// TIA Portal V20 export
// export: Created 2025-12-01T14:57:06.1512195Z, ExportSetting None, DisplayName Totally Integrated Automation Portal, DisplayVersion V20 Update 3, DisplayName TIA Portal Openness, DisplayVersion V20 Update 3, DisplayName TIA Portal Version Control Interface, DisplayVersion V20 Update 3, DisplayName STEP 7 Professional, DisplayVersion V20 Update 3, DisplayName STEP 7 Safety, DisplayVersion V20 Update 2, DisplayName WinCC Basic/Comfort/Advanced, DisplayVersion V20 Update 3, DisplayName WinCC Professional, DisplayVersion V20 Update 3, DisplayName WinCC Unified, DisplayVersion V20 Update 3
FUNCTION "FC903_Tratamiento_MesasDeZona" : Void   // FC903, STL
{ S7_Optimized_Access := 'FALSE' }
// stored: AutoNumber false
   VAR_INPUT
      NumZona : UInt;
   END_VAR
   VAR_IN_OUT
      MesasDeZona : "InternasDeLaZona";
   END_VAR
   VAR_TEMP
      Zona : UInt;
      Mesa : UInt;
      MaxMesas : UInt;
      MesasParo : Bool;
      MesasBlando : Bool;
      MesasManual : Bool;
      MesasError : Bool;
      MesasTodasParo : Bool;
      MesasTodasManual : Bool;
   END_VAR
BEGIN

NETWORK
TITLE = Inicializacion
/////////////////////////////////////////////////////////////////////////////
/////////////////////////////////////////////////////////////////////////////
// --- Tareas Iniciales

      L     #NumZona;  // - Numero de Zana
      T     #Zona;

      L     #Zona;  // Es el CCPIF ?
      L     0;
      <>I;
      JC    CBOX;
      JU    CBOX;  // Para Tramiento el CBOX y CCPIF el mismo

/////////////////////////////////////////////////////////////////////////////
/////////////////////////////////////////////////////////////////////////////
// Es de Tipo CCPIF
CCPIF:NOP   0;
      SET;  // - Inicializar Variables Internas
      R     #MesasParo;  //   Para el CCPIF
      R     #MesasBlando;
      R     #MesasManual;
      R     #MesasError;
      R     #MesasTodasParo;
      R     #MesasTodasManual;
      JU    Final;  //   Finaliza para CCPIF


/////////////////////////////////////////////////////////////////////////////
/////////////////////////////////////////////////////////////////////////////
// Es de tipo CBOX
CBOX: NOP   0;

      SET;  // - Inicializar Variables Internas
      R     #MesasParo;  //   Para un CBOX
      R     #MesasBlando;
      R     #MesasManual;
      R     #MesasError;
      S     #MesasTodasParo;
      S     #MesasTodasManual;


/////////////////////////////////////////////////////////////////////////////
/////////////////////////////////////////////////////////////////////////////
// --- Datos iniciales de Trabajo

      L     "CTE_MaxMesas";  // - Numero Max. de Mesas en el PLC
      T     #MaxMesas;



NETWORK
TITLE = Tratamiento
/////////////////////////////////////////////////////////////////////////////
/////////////////////////////////////////////////////////////////////////////
// ---  Tratamiento del Estado de las Mesas que pertenecn a la Mesa

      L     1;  // Inicializar
      T     #Mesa;
InicioBucle:NOP   0;

      SET;  //    Zona 0
      L     "DB914_Conf_Mesas_DeZona".MesasDeZona[#Mesa, 0].ZonaPerteneceMesa;
      L     #Zona;
      ==I;
      JC    MesaEncontrada;

      SET;  //    Zona 1
      L     "DB914_Conf_Mesas_DeZona".MesasDeZona[#Mesa, 1].ZonaPerteneceMesa;
      L     #Zona;
      ==I;
      JC    MesaEncontrada;

      SET;  //    Zona 2
      L     "DB914_Conf_Mesas_DeZona".MesasDeZona[#Mesa, 2].ZonaPerteneceMesa;
      L     #Zona;
      ==I;
      JC    MesaEncontrada;

      SET;  //    Zona 3
      L     "DB914_Conf_Mesas_DeZona".MesasDeZona[#Mesa, 3].ZonaPerteneceMesa;
      L     #Zona;
      ==I;
      JC    MesaEncontrada;

      SET;  //    Zona 4
      L     "DB914_Conf_Mesas_DeZona".MesasDeZona[#Mesa, 4].ZonaPerteneceMesa;
      L     #Zona;
      ==I;
      JC    MesaEncontrada;

      JU    ContinuarBucle;


/////////////////////////////////////////////////////////////////////////////
/////////////////////////////////////////////////////////////////////////////
// --- Comprobacion del Estado Zona de la Mesa
MesaEncontrada:NOP   0;

      SET;  // - Alguna mesa en Error
      A     "DB902_Estado_ZonaMesa".EstadoMesas[#Mesa].Error_CBx;
      S     #MesasError;

      SET;  // - Alguna mesa en Paro
      AN    "DB902_Estado_ZonaMesa".EstadoMesas[#Mesa].Marcha_CBx;
      S     #MesasParo;

      SET;  // - Alguna mesa en ParoBlando
      A     "DB902_Estado_ZonaMesa".EstadoMesas[#Mesa].ParoBlando_CBx;
      S     #MesasBlando;

      SET;  // - Alguna mesa en Manual
      AN    "DB902_Estado_ZonaMesa".EstadoMesas[#Mesa].Automatico_CBx;
      S     #MesasManual;

      SET;  // - Todas las mesas en Paro
      A     "DB902_Estado_ZonaMesa".EstadoMesas[#Mesa].Marcha_CBx;
      R     #MesasTodasParo;

      SET;  // - Todas las mesas en Manual
      A     "DB902_Estado_ZonaMesa".EstadoMesas[#Mesa].Automatico_CBx;
      R     #MesasTodasManual;


/////////////////////////////////////////////////////////////////////////////
/////////////////////////////////////////////////////////////////////////////
// --- Comprobacion del Estado Zona de la Maquina

      SET;  // - Alguna Maquina en Error
      A     "DB903_Estado_ZonaMaquina".EstadoMaquina[#Mesa].Error_CBx;
      S     #MesasError;

/////////////////////////////////////////////////////////////////////////////
/////////////////////////////////////////////////////////////////////////////
// --- Es Final del Tratamiento
ContinuarBucle:NOP   0;

      L     #MaxMesas;  // - Final del Numero de Mesas ?
      L     #Mesa;
      <=I;
      JC    FinBucle;

      L     #Mesa;  // - Incrementa a la siguiente Mesa
      L     1;
      +I;
      T     #Mesa;

      JU    InicioBucle;  // - Siguiente Mesa

// --------------------------------------------------------------------------------------------------
// --------------------------------------------------------------------------------------------------
// --- Final del Tratmiento

FinBucle:NOP   0;


NETWORK
TITLE = Final
// --------------------------------------------------------------------------------------------------
// --------------------------------------------------------------------------------------------------
// --- Tareas finales

Final:NOP   0;
// --------------------------------------------------------------------------------------------------
// --------------------------------------------------------------------------------------------------
// --- Activacion de las Salidas

      A     #MesasParo;
      =     #MesasDeZona.MesasParo;

      A     #MesasBlando;
      =     #MesasDeZona.MesasBlando;

      A     #MesasManual;
      =     #MesasDeZona.MesasManual;

      A     #MesasError;
      =     #MesasDeZona.MesasError;

      A     #MesasTodasParo;
      =     #MesasDeZona.MesasTodasParo;

      A     #MesasTodasManual;
      =     #MesasDeZona.MesasTodasManual;


END_FUNCTION
